{attribute 'GeneratedUsingTerminal: KL3356'}
{attribute addProperty BoxType "KL3356"}
{attribute addProperty Id "StatusAT %I*USINT0RegInAT %I*UINT0AnStatusAT %I*USINT0WeightAT %I*UINT0CtrlAT %Q*USINT0RegOutAT %Q*UINT0AnCtrlAT %Q*USINT0"}
{attribute addProperty CRC "1318919725"}
{attribute addProperty Size "0"}
TYPE Channel_4E9D1E2D :
STRUCT
	{attribute addProperty Name "Status"}
	Status AT %I* : USINT;
	{attribute addProperty Name "RegIn"}
	RegIn AT %I* : UINT;
	{attribute addProperty Name "AnStatus"}
	AnStatus AT %I* : USINT;
	{attribute addProperty Name "Weight"}
	Weight AT %I* : UINT;
	{attribute addProperty Name "Ctrl"}
	Ctrl AT %Q* : USINT;
	{attribute addProperty Name "RegOut"}
	RegOut AT %Q* : UINT;
	{attribute addProperty Name "AnCtrl"}
	AnCtrl AT %Q* : USINT;
END_STRUCT
END_TYPE

(* stored: Version 1.2.0.0, ProductVersion 3.1.4024.11
   DUT Channel_4E9D1E2D: Id {f494fc30-d72f-4512-84a8-9f1551b535c3} *)
